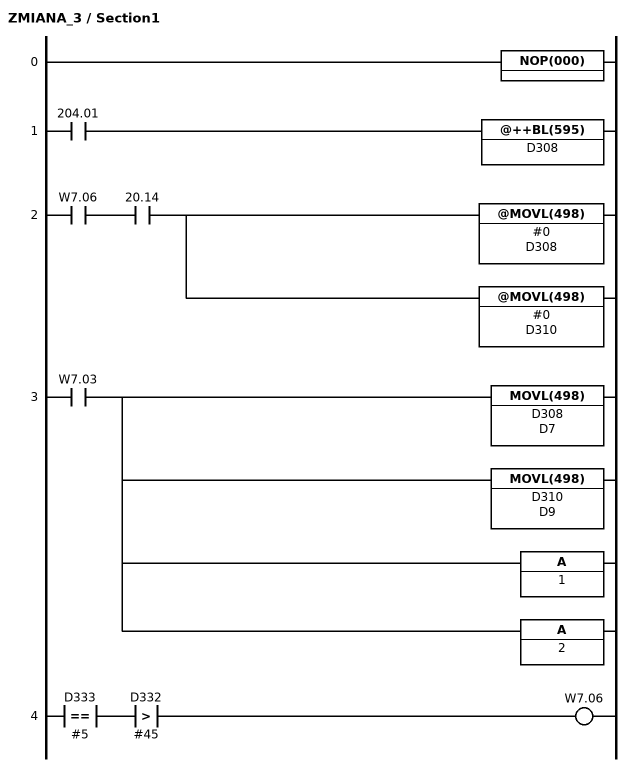
; [picture p96: ZMIANA_3 / Section1, rungs 0-4]
; rung 0
NOP(000)
; rung 1
LD 204.01
@++BL(595) D308
; rung 2
LD W7.06
AND 20.14
@MOVL(498) #0 D308
@MOVL(498) #0 D310
; rung 3
LD W7.03
MOVL(498) D308 D7
MOVL(498) D310 D9  // 
A  1
A  2
// 
// 
; rung 4
LD=(300) D333 #5
AND>(320) D332 #45
OUT W7.06
; rung 5
END(001)